// TwinCAT 3 PLC project Palletizer
// ProgramVersion: 3.1.4023.0
// libraries:
//   MqttFramework, * (FactoryAutomation)
//   StateMachineLib, * (FactoryAutomation)
//   StepWorkerLib, * (FactoryAutomation)
//   Tc2_Standard, * (Beckhoff Automation GmbH)
//   Tc2_System, * (Beckhoff Automation GmbH)
//   Tc3_Module, * (Beckhoff Automation GmbH)
// project tree:
//   Basic/ A_Actuator.TcPOU
//   Basic/Conveyors/ Conveyor.TcPOU, PalletizerConveyor.TcPOU
//   Basic/Cylinder/ Cylinder.TcPOU
//   Basic/Elevator/ Elevator.TcPOU, PalletizerElevator.TcPOU
//   Basic/Sensor/ Sensor.TcPOU
//   / PlcTask.TcTTO
//   POUs/ MAIN.TcPOU, Palletizer.TcPOU
//   POUs/RemoteControl/ E_ActuatorCmdType.TcDUT, E_ActuatorType.TcDUT, E_ModeType.TcDUT, PalletizerRemoteCtrl.TcPOU
// real-time tasks:
//   TASK PlcTask: cycle T#10ms, priority 20, ADS port 350

CONFIGURATION Palletizer
    RESOURCE PLC ON TwinCAT3
        TASK PlcTask(INTERVAL := T#10ms, PRIORITY := 20);
        PROGRAM MAIN WITH PlcTask : MAIN;
        PROGRAM ADS WITH PlcTask : ADS;
    END_RESOURCE
END_CONFIGURATION

// ---- POUs/RemoteControl/E_ActuatorCmdType.TcDUT

TYPE E_ActuatorCmdType :
(
	eNO_ACTUATOR_CMD := 0,
	eFORWARD,
	eBACKWARD,
	eVELOCITY,
	ePUSH,
	eRETRACT,
	eUP,
	eDOWN,
	eUP_TO_LIMIT,
	eDOWN_TO_LIMIT,
	eSTART,
	eSTOP,
	eHOME,
	eRESET
)UINT;
END_TYPE
(*
			+	mode manual
			
				+	actuator type
				
					+	Belt
						+	forware
						+	backward
						
					+	Chain
						+	forward
						+	backward	
						
					+	BeltConveyor
						+	forward
						+	backward
						+	velocity
						
					+	RollerConveyor
						+	forward
						+	backward
						+	velocity	
						
					+	Turn
						+	forward
						+	backward
						
					+	Clamper
						+	clamp
						+	unclamp
	
					+	Pusher
						+	push forward
						+	push backward
						
					+	Plate
						+	open plate
						+	close plate
						
					+	Elevator
						+	up
						+	down
						+	to limit
						
			+	mode automatic
				
				+	start
				+	stop
			
			+	mode system
			
				+	home
				+	reset
				*)

// ---- POUs/RemoteControl/E_ActuatorType.TcDUT

TYPE E_ActuatorType :
(
	eNO_ACTUATOR := 0,
	ePALLETIZER_BELT,
	ePALLETIZER_CHAIN,
	eBELT_CONVEYOR,
	eROLLER_CONVEYOR,
	eTURN_CYLINDER,
	eCLAMPER_CYLINDER,
	ePUSHER_CYLINDER,
	ePLATE_CYLINDER,
	eELEVATOR
)UINT;

END_TYPE
(*
+	mode manual
			
				+	actuator type
				
					+	Belt
						+	forware
						+	backward
						
					+	Chain
						+	forward
						+	backward	
						
					+	BeltConveyor
						+	forward
						+	backward
						+	velocity
						
					+	RollerConveyor
						+	forward
						+	backward
						+	velocity	
						
					+	Turn
						+	forward
						+	backward
						
					+	Clamper
						+	clamp
						+	unclamp
	
					+	Pusher
						+	push forward
						+	push backward
						
					+	Plate
						+	open plate
						+	close plate
						
					+	Elevator
						+	up
						+	down
						+	to limit
						
			+	mode automatic
				
				+	start
				+	stop
			
			+	mode system
			
				+	home
				+	reset
				*)

// ---- POUs/RemoteControl/E_ModeType.TcDUT

TYPE E_ModeType :
(
	eNO_MODE_TYPE := 0,
	eAUTOMATIC_MODE_TYPE,
	eMANUAL_MODE_TYPE,
	eSYSTEM_MODE_TYPE
)UINT;
END_TYPE

// ---- POUs/MAIN.TcPOU
PROGRAM MAIN
VAR
	fbRemoteControl : PalletizerRemoteCtrl;
	fbPalletizer : Palletizer;
END_VAR

fbPalletizer();
fbRemoteControl(fbPalletizer := fbPalletizer);

END_PROGRAM

// ---- POUs/RemoteControl/PalletizerRemoteCtrl.TcPOU
FUNCTION_BLOCK PalletizerRemoteCtrl
VAR_INPUT
	bExecute : BOOL;
END_VAR
VAR_IN_OUT
	fbPalletizer : Palletizer;
END_VAR
VAR_OUTPUT
END_VAR
VAR
	
	udiStep : UDINT;
	messageIndex : UINT;
	remoteCtrlPayload : ST_MqttPayload;
	
	eActuatorType : E_ActuatorType;

END_VAR

(*

Description:
========================================================================	
	
	+	check if AdsConnector is connected
	+	if connected, subscribe to PalHmi topic
	+	check for incoming messages
	+	if message available, check message type 
	+	possible message types are:
	
			+	mode manual
			
				+	actuator type
				
					+	Belt
						+	forware
						+	backward
						
					+	Chain
						+	forward
						+	backward	
						
					+	BeltConveyor
						+	forward
						+	backward
						+	velocity
						
					+	RollerConveyor
						+	forward
						+	backward
						+	velocity	
						
					+	Turn
						+	forward
						+	backward
						
					+	Clamper
						+	clamp
						+	unclamp
	
					+	Pusher
						+	push forward
						+	push backward
						
					+	Plate
						+	open plate
						+	close plate
						
					+	Elevator
						+	up
						+	down
						+	to limit
						
			+	mode automatic
				
				+	start
				+	stop
			
			+	mode system
			
				+	home
				+	reset
				
			
=========================================================================

*)



IF 	ADS.fbAdsConnector.isConnected
	AND bExecute
THEN

	udiStep := 10;
ELSE
	udiStep := 0;
END_IF

CASE udiStep OF

	10:
		IF ADS.fbMqttClient.subscribe('PalHmi',THIS)
		THEN
			udiStep := 20;
		END_IF
		
	20:
		messageIndex := ADS.fbMqttClient.isNewMessage('PalHmi');
		IF messageIndex > 0
		THEN
		
			evaluateMode(Ads.fbMqttClient.getNewMessage(messageIndex));
			
		END_IF
			
		
END_CASE

METHOD PRIVATE evaluateActuator : BOOL
VAR_INPUT
	remoteCtrlPayload : ST_MqttPayload;
END_VAR
VAR
	eCmd : E_ActuatorCmdType;
	eActuator : E_ActuatorType;
END_VAR
eActuator := BYTE_TO_UINT(remoteCtrlPayload.data[2]);
eCmd := BYTE_TO_UINT(remoteCtrlPayload.data[3]);

CASE eActuator OF

	ePALLETIZER_BELT:
		
		fbPalletizer.fbBeltConveyor.cmd := eCmd;
		
	ePALLETIZER_CHAIN:
	
		fbPalletizer.fbPalletizerChain.cmd := eCmd;
		
	eBELT_CONVEYOR:
		
		fbPalletizer.fbBeltConveyor.cmd := eCmd;
		
	eROLLER_CONVEYOR:
		
		fbPalletizer.fbRollerConveyor.cmd := eCmd;
		
	eTURN_CYLINDER:
		
		fbPalletizer.fbTurnCylinder.cmd := eCmd;
	
	eCLAMPER_CYLINDER:
		
		fbPalletizer.fbClamperCylinder.cmd := eCmd;
	
	ePUSHER_CYLINDER:
		
		fbPalletizer.fbPusherCylinder.cmd := eCmd;
	
	ePLATE_CYLINDER:
		
		fbPalletizer.fbPlateCylinder.cmd := eCmd;
		
	eELEVATOR:
	
		fbPalletizer.fbElevator.cmd := eCmd;
	
END_CASE
END_METHOD

METHOD PRIVATE evaluateMode : BOOL
VAR_INPUT
	remoteCtrlPayload : ST_MqttPayload;
END_VAR
VAR	
	eCmd : E_ActuatorCmdType;
	eMode : E_ModeType;
END_VAR
(*
	data : ARRAY[1..32] OF Byte;
	
	data[1] -> mode type
	data[2] -> actutator type
	data[3] -> cmd
*)

eMode := BYTE_TO_UINT(remoteCtrlPayload.data[1]);
eCmd := BYTE_TO_UINT(remoteCtrlPayload.data[3]);

CASE eMode OF

	eAUTOMATIC_MODE_TYPE,
	eSYSTEM_MODE_TYPE:
		fbPalletizer.cmd := eCmd;
	eMANUAL_MODE_TYPE:
		evaluateActuator(remoteCtrlPayload);
	
END_CASE
END_METHOD

END_FUNCTION_BLOCK

// ---- POUs/Palletizer.TcPOU
FUNCTION_BLOCK Palletizer EXTENDS A_Actuator
VAR_INPUT
	fbBeltConveyor : Conveyor;
	fbPalletizerChain : Conveyor;
	fbRollerConveyor : Conveyor;
	fbTurnCylinder : Cylinder;
	fbClamperCylinder : Cylinder;
	fbPusherCylinder : Cylinder;
	fbPlateCylinder : Cylinder;
	fbElevator : Elevator; 
END_VAR
VAR_OUTPUT
	
END_VAR
VAR

END_VAR

END_FUNCTION_BLOCK

// ---- Basic/A_Actuator.TcPOU
FUNCTION_BLOCK ABSTRACT A_Actuator
VAR_INPUT
	
END_VAR
VAR_OUTPUT
END_VAR
VAR
	eCmd : E_ActuatorCmdType;
	
END_VAR

PROPERTY cmd : E_ActuatorCmdType
GET
cmd := eCmd;
END_GET
SET
eCmd := cmd;
executeCmd();
END_SET
END_PROPERTY

METHOD ABSTRACT executeCmd : BOOL
VAR_INPUT
	
END_VAR
END_METHOD

END_FUNCTION_BLOCK

// ---- Basic/Conveyors/Conveyor.TcPOU
FUNCTION_BLOCK Conveyor EXTENDS A_Actuator
VAR_INPUT
END_VAR

VAR_OUTPUT
	bStart  : BOOL;
END_VAR
VAR
	
	fbStart : BoolOut;
END_VAR

bStart := fbStart.getValue;

{warning 'Eigenschaftenimplementierung hinzufügen'}
PROPERTY cmd : E_ActuatorCmdType
GET
END_GET
SET
END_SET
END_PROPERTY

PROPERTY getStart : I_StepCondition
GET
getStart := fbStart;
END_GET
END_PROPERTY

METHOD Off : BOOL
VAR_INPUT
END_VAR
fbStart.setValue := FALSE;
END_METHOD

METHOD On : BOOL
VAR_INPUT
END_VAR
fbStart.setValue := TRUE;
END_METHOD

END_FUNCTION_BLOCK

// ---- Basic/Cylinder/Cylinder.TcPOU
FUNCTION_BLOCK Cylinder EXTENDS A_Actuator
VAR_INPUT
END_VAR
VAR_OUTPUT
	bExtended : BOOL;
	bExtend : BOOL;
END_VAR
VAR
	fbExtendedSignal : BoolIn;
	fbExtend : BoolOut;
END_VAR

bExtended := fbExtendedSignal.getValue;
bExtend := fbExtend.getValue;

{warning 'Eigenschaftenimplementierung hinzufügen'}
PROPERTY cmd : E_ActuatorCmdType
GET
END_GET
SET
END_SET
END_PROPERTY

METHOD Extend : BOOL
VAR_INPUT
END_VAR
fbExtend.setValue := TRUE;
END_METHOD

PROPERTY getExtend : I_StepCondition
GET
getExtend := fbExtend;
END_GET
END_PROPERTY

METHOD Retract : BOOL
VAR_INPUT
END_VAR
fbExtend.setValue := FALSE;
END_METHOD

END_FUNCTION_BLOCK

// ---- Basic/Elevator/Elevator.TcPOU
FUNCTION_BLOCK Elevator EXTENDS A_Actuator
VAR_INPUT
END_VAR
VAR_OUTPUT
END_VAR
VAR
END_VAR

{warning 'Eigenschaftenimplementierung hinzufügen'}
PROPERTY cmd : E_ActuatorCmdType
GET
END_GET
SET
END_SET
END_PROPERTY

END_FUNCTION_BLOCK

// ---- Basic/Conveyors/PalletizerConveyor.TcPOU
FUNCTION_BLOCK PalletizerConveyor EXTENDS Conveyor
VAR_INPUT
END_VAR
VAR_OUTPUT
	bStartBackward : BOOL;
END_VAR
VAR	
	fbStartBackward : BoolOut;
END_VAR

SUPER^();
bStartBackward := fbStartBackward.getValue;

PROPERTY getStartBackward : I_StepCondition
GET
getStartBackward := fbStartBackward;
END_GET
END_PROPERTY

END_FUNCTION_BLOCK

// ---- Basic/Elevator/PalletizerElevator.TcPOU
FUNCTION_BLOCK PalletizerElevator EXTENDS Elevator
VAR_INPUT
END_VAR
VAR_OUTPUT
	isMoving : BOOL;
END_VAR
VAR
	fbElevatorMoving : Sensor;
	fbElevatorUp : BoolOut;
	fbElevatorDown : BoolOut;
	fbElevatorToLimit : BoolOut;
END_VAR

isMoving := fbElevatorMoving.bSignal;

PROPERTY getElevatorMoving : I_StepCondition
GET
getElevatorMoving := fbElevatorMoving.getSignal;
END_GET
END_PROPERTY

METHOD MoveDown : BOOL
VAR_INPUT
END_VAR
fbElevatorDown.setValue := TRUE;
fbElevatorUp.setValue := FALSE;

fbElevatorToLimit.setValue := TRUE;
END_METHOD

METHOD MoveUp : BOOL
VAR_INPUT
END_VAR
fbElevatorUp.setValue := TRUE;
fbElevatorDown.setValue := FALSE;

fbElevatorToLimit.setValue := TRUE;
END_METHOD

END_FUNCTION_BLOCK

// ---- Basic/Sensor/Sensor.TcPOU
FUNCTION_BLOCK Sensor
VAR_INPUT
END_VAR
VAR_OUTPUT
	bSignal  : BOOL;
END_VAR
VAR
	fbSignal : BoolIn;
END_VAR

bSignal := fbSignal.getValue;

PROPERTY getSignal : I_StepCondition
GET
getSignal := fbSignal;
END_GET
END_PROPERTY

END_FUNCTION_BLOCK
